SUBAPPLICATION PublishEventOpcUaFull (* Publish Event using OpcUa. All possible parameters are available to be set *)
  (* Standard: 61499-2; Description: Copyright (c) 2019 fortiss GmbH This program and the accompanying materials are made SPDX-License-Identifier: EPL-2.0 *)
  (* Version 1.0, 2019-11-12, Jose Cabral, fortiss GmbH *)
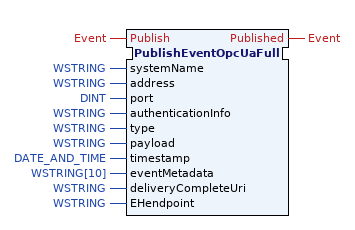
  EVENT_INPUT
    Publish;
  END_EVENT
  EVENT_OUTPUT
    Published;
  END_EVENT
  VAR_INPUT
    systemName : WSTRING; (* Identification of the system *)
    address : WSTRING; (* Address of the offered services *)
    port : DINT; (* Port of the of the offered services *)
    authenticationInfo : WSTRING; (* Authentication info of the system *)
    type : WSTRING; (* The type of the event, an event ID of sorts *)
    payload : WSTRING; (* String data of the event *)
    timestamp : DATE_AND_TIME; (* Date and time of the event *)
    eventMetadata : ARRAY [0..9] OF WSTRING; (* Key=value pairs of additional data about the event *)
    deliveryCompleteUri : WSTRING; (* The URL subpath the Event Handler can use to inform the publisher about the results of the event propagation. If null, the Event Handler will not try to send the results *)
    EHendpoint : WSTRING; (* Endpoint (IP:PORT/URI) of the Event Handler (not officially in the documentation, but it simplifies the FBs) *)
  END_VAR
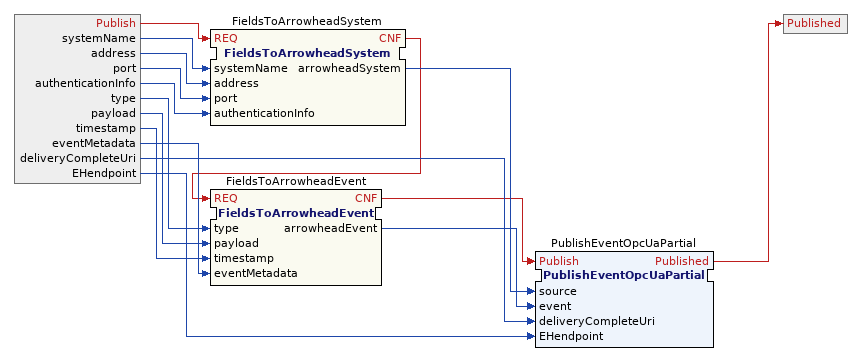
  FBS
    FieldsToArrowheadEvent : FieldsToArrowheadEvent;
    FieldsToArrowheadSystem : FieldsToArrowheadSystem;
  END_FBS
  SUBAPPS
    PublishEventOpcUaPartial : PublishEventOpcUaPartial;
  END_SUBAPPS
  EVENT_CONNECTIONS
    FieldsToArrowheadSystem.CNF TO FieldsToArrowheadEvent.REQ;
    Publish TO FieldsToArrowheadSystem.REQ;
    FieldsToArrowheadEvent.CNF TO PublishEventOpcUaPartial.Publish;
    PublishEventOpcUaPartial.Published TO Published;
  END_CONNECTIONS
  DATA_CONNECTIONS
    systemName TO FieldsToArrowheadSystem.systemName;
    address TO FieldsToArrowheadSystem.address;
    port TO FieldsToArrowheadSystem.port;
    authenticationInfo TO FieldsToArrowheadSystem.authenticationInfo;
    type TO FieldsToArrowheadEvent.type;
    payload TO FieldsToArrowheadEvent.payload;
    timestamp TO FieldsToArrowheadEvent.timestamp;
    eventMetadata TO FieldsToArrowheadEvent.eventMetadata;
    FieldsToArrowheadSystem.arrowheadSystem TO PublishEventOpcUaPartial.source;
    FieldsToArrowheadEvent.arrowheadEvent TO PublishEventOpcUaPartial.event;
    deliveryCompleteUri TO PublishEventOpcUaPartial.deliveryCompleteUri;
    EHendpoint TO PublishEventOpcUaPartial.EHendpoint;
  END_CONNECTIONS
END_SUBAPPLICATION
